_CFC_ (* Continuous Function Chart, elements in execution order *)
#0 INT_TO_REAL(SHU6_P2_TE6_AI1)
#1 DIV(#0, 10)
#2 SHU6_P2_TE6_T_VN <= #1
#3 I_GT_TE6:ISTOK_GT(dost: TRUE, x: #1, ust: SHU6_P2_TE6_HIGHLIMIT, shkal: -, gist: 1)
#4 SUB(SHU6_P2_TE6_T_UST, 0.6)
#5 I_LT_TE6:ISTOK_LT(dost: TRUE, x: #1, ust: SHU6_P2_TE6_LOWLIMIT, shkal: -, gist: 1)
#6 OR(#3.Xb, #5.Xm)
#7 TON_DOST:TON(IN: NOT #6, PT: T#10s)
#8 SHU6_P2_TE6_T_DOST <= #7.Q
#9 fb_TE6_m_UST:ISTOK_LT(dost: #7.Q, x: #1, ust: #4, shkal: -, gist: 0.5)
#10 SHU6_P2_TE6_TE_M_UST <= #9.Xm
#11 SHU6_P2_TE6_TE_NM_UST <= #9.XmN
#12 ADD(SHU6_P2_TE6_T_UST, 0.6)
#13 fb_TE6_b_UST:ISTOK_GT(dost: #7.Q, x: #1, ust: #12, shkal: -, gist: 0.5)
#14 SHU6_P2_TE6_TE_B_UST <= #13.Xb
#15 SHU6_P2_TE6_TE_NB_UST <= #13.XbN
_END_CFC_
(* the same logic as Structured Text *)
_t108 := INT_TO_REAL(SHU6_P2_TE6_AI1) / 10;
SHU6_P2_TE6_T_VN := _t108;
I_GT_TE6(dost := TRUE, x := _t108, ust := SHU6_P2_TE6_HIGHLIMIT, gist := 1);
I_LT_TE6(dost := TRUE, x := _t108, ust := SHU6_P2_TE6_LOWLIMIT, gist := 1);
TON_DOST(IN := NOT (I_GT_TE6.Xb OR I_LT_TE6.Xm), PT := T#10s);
SHU6_P2_TE6_T_DOST := TON_DOST.Q;
fb_TE6_m_UST(dost := TON_DOST.Q, x := _t108, ust := SHU6_P2_TE6_T_UST - 0.6, gist := 0.5);
SHU6_P2_TE6_TE_M_UST := fb_TE6_m_UST.Xm;
SHU6_P2_TE6_TE_NM_UST := fb_TE6_m_UST.XmN;
fb_TE6_b_UST(dost := TON_DOST.Q, x := _t108, ust := SHU6_P2_TE6_T_UST + 0.6, gist := 0.5);
SHU6_P2_TE6_TE_B_UST := fb_TE6_b_UST.Xb;
SHU6_P2_TE6_TE_NB_UST := fb_TE6_b_UST.XbN;
END_PROGRAM

(* POU Lib/ISTOK_EQ, CFC *)
FUNCTION_BLOCK ISTOK_EQ
VAR_INPUT
	dost: BOOL;
	X: REAL;
	ust: REAL;
	shkal: REAL;
	gist: REAL;
END_VAR
VAR_OUTPUT
	Xeq: BOOL;
	Xneq: BOOL;
END_VAR
VAR
END_VAR
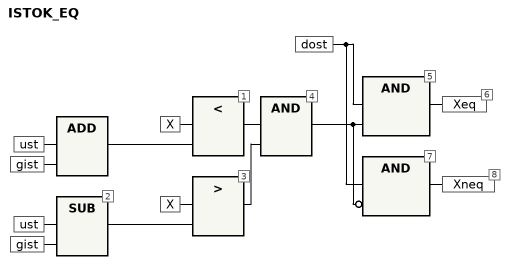
_CFC_ (* Continuous Function Chart, elements in execution order *)
#0 ADD(ust, gist)
#1 <(X, #0)
#2 SUB(ust, gist)
#3 >(X, #2)
#4 AND(#1, #3)
#5 AND(dost, #4)
#6 Xeq <= #5
#7 AND(dost, NOT #4)
#8 Xneq <= #7
_END_CFC_
END_FUNCTION_BLOCK

(* POU Input/AI/YA3_POS, CFC *)
PROGRAM YA3_POS
VAR
	ofset: REAL;
	fb_YA3: ISTOK_ANALOGVH;
	Lt_otkr_zakr: ISTOK_LT;
	gt_otkr_otr: ISTOK_GT;
	fb_YA3bUST_VKL_STER_REG: ISTOK_GT;
	fb_YA3mOTKL_STER_REG: ISTOK_LT;
END_VAR
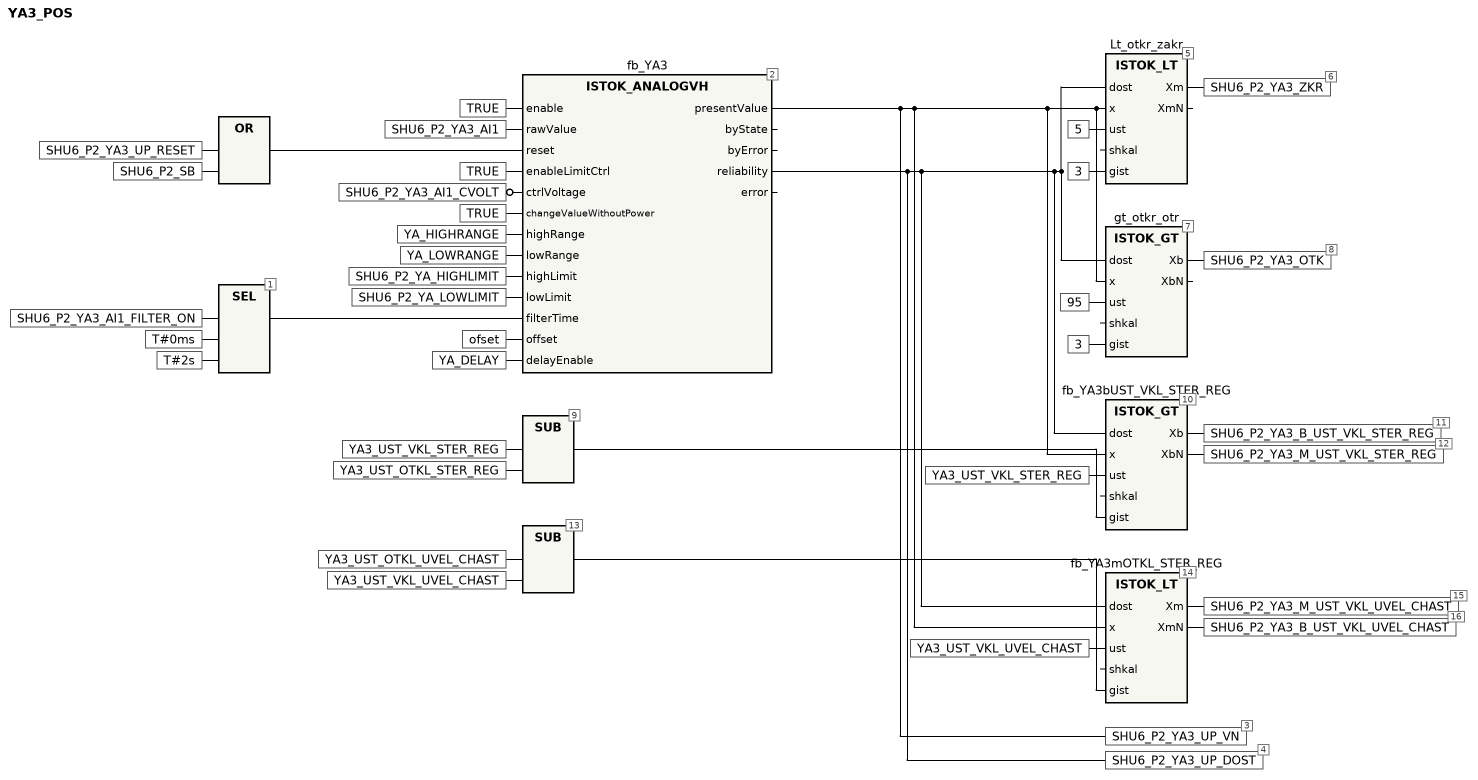
